// TIA Portal V17 export
// export: Created 2026-04-13T11:12:43.5748285Z, ExportSetting WithDefaults, DisplayName Totally Integrated Automation Portal, DisplayVersion V17 Update 4, DisplayName TIA Portal Openness, DisplayVersion V17 Update 4, DisplayName TIA Portal Version Control Interface, DisplayVersion V17, DisplayName SINAMICS Startdrive Advanced, DisplayVersion V17, DisplayName SINAMICS Startdrive G130, G150, S120, S150, SINAMICS MV, S210, DisplayVersion V17, DisplayName SINAMICS Startdrive G110M, G120, G120C, G120D, G120P, G115D, DisplayVersion V17, DisplayName STEP 7 Professional, DisplayVersion V17 Update 4, DisplayName STEP 7 Safety, DisplayVersion V17, DisplayName WinCC Professional, DisplayVersion V17 Update 4
FUNCTION_BLOCK "31-温度控制"   // FB21, LAD
{ S7_Optimized_Access := 'FALSE' }
VERSION : 0.1
// stored: AutoNumber true, IsIECCheckEnabled false, SetENOAutomatically false, UDAEnableTagReadback false
   VAR_IN_OUT
      进温设定 : Real;
      加热器开关 : Bool;
      自整定开关 : Bool;
      进温读 : Real;
      出温读 : Real;
      尾温读 : Real;
      进风温度P : Real;
      进风温度I : Real;
      进风温度D : Real;
      JF进风温度写读 : Real;
   END_VAR
   VAR DB_SPECIFIC
      CTU { S7_SetPoint := 'True'} : CTU_INT;
      TEMP { S7_SetPoint := 'True'} : Bool;
      TP : Array[0..40] of Bool;
      T1_PV_读 : Int;
      T2_PV_读 : Int;
      T3_PV_读 : Int;
      T4_PV_读 : Int;
      T5_PV_读 : Int;
      T1_SV_写 : Int;
      T1_P值比对1 : Int;
      T1_P值比对2 : Int;
      ST1 : Real;
      ST2 : Real;
      ST3 : Real;
      ST4 : Real;
      ST5 : Real;
      ST16 : Real;
      ST17 : Real;
      ST18 : Real;
      ST20 : Real;
      ST21 : Real;
      ST22 : Real;
      进温P读 : Int;
      进温I读 : Int;
      进温D读 : Int;
      T1_P_I_D_读 : Array[0..2] of Int;
      IEC_Timer_0_Instance { S7_SetPoint := 'True'} : TON_TIME;
      JF进风温度写读辅 { S7_SetPoint := 'True'} : Int;
      进温AT_写 : Int;
      进温AT_读 : Int;
      自整定开关字 : Int;
      加热器开关字 : Int;
   END_VAR
   VAR
      Modbus_Comm_Load_Instance { S7_SetPoint := 'True'} : Modbus_Comm_Load;
      Modbus_Master { S7_SetPoint := 'True'} : Modbus_Master;
   END_VAR
   VAR_TEMP   // added for the SCL form of the ladder/FBD networks
      _w1 : Bool;
      _w2 : Bool;
      _w3 : Bool;
      _w4 : Bool;
   END_VAR
BEGIN

REGION Network 1
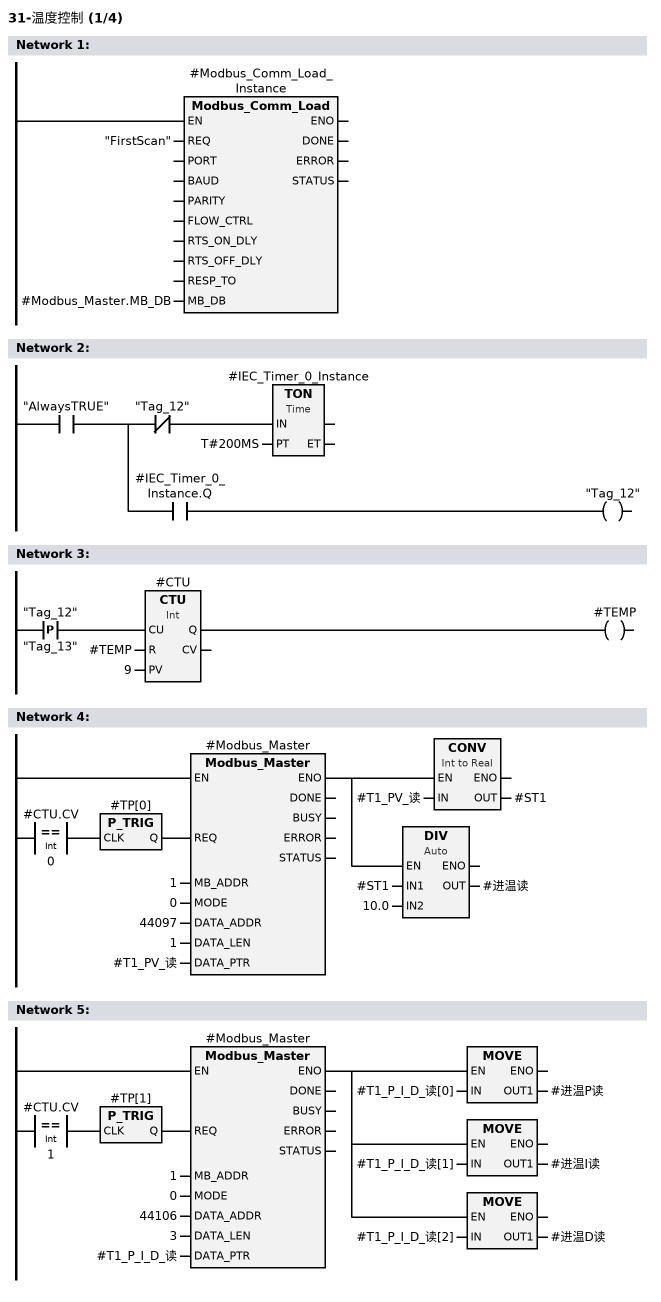
   RUNG wire#powerrail
      #Modbus_Comm_Load_Instance.Modbus_Comm_Load(REQ := "FirstScan", PORT :=, BAUD :=, PARITY :=, FLOW_CTRL :=, RTS_ON_DLY :=, RTS_OFF_DLY :=, RESP_TO :=, MB_DB := #Modbus_Master.MB_DB, DONE =>, ERROR =>, STATUS =>)
   END_RUNG
   // the same network as SCL:
   #Modbus_Comm_Load_Instance(REQ := "FirstScan", MB_DB := #Modbus_Master.MB_DB);   // Modbus_Comm_Load
END_REGION

REGION Network 2
   RUNG wire#powerrail
      Contact( "AlwaysTRUE" )
      wire#w1
      I_Contact( "Tag_12" )
      { S7_Templates := "time_type := Time" } #IEC_Timer_0_Instance.TON(pt := T#200MS, et =>)
   END_RUNG
   RUNG wire#w1
      Contact( #IEC_Timer_0_Instance.Q )
      Coil( "Tag_12" )
   END_RUNG
   // the same network as SCL:
   #IEC_Timer_0_Instance(IN := "AlwaysTRUE" AND NOT "Tag_12", PT := T#200MS);   // TON
   "Tag_12" := "AlwaysTRUE" AND #IEC_Timer_0_Instance.Q;
END_REGION

REGION Network 3
   RUNG wire#powerrail
      P_Contact(operand := "Tag_12", bit := "Tag_13")
      { S7_Templates := "value_type := Int" } #CTU.CTU(r := #TEMP, pv := 9, cv =>)
      Coil( #TEMP )
   END_RUNG
   // the same network as SCL:
   #_w1 := "Tag_12" AND NOT "Tag_13";   // rising edge of "Tag_12"
   "Tag_13" := "Tag_12";
   #CTU(CU := #_w1, R := #TEMP, PV := 9);   // CTU
   #TEMP := #CTU.Q;
END_REGION

REGION Network 4
   RUNG wire#powerrail
      #Modbus_Master.Modbus_Master(REQ := wire#w1, MB_ADDR := 1, MODE := 0, DATA_ADDR := 44097, DATA_LEN := 1, DATA_PTR := #T1_PV_读, DONE =>, BUSY =>, ERROR =>, STATUS =>)
      wire#w2
      { S7_Templates := "[SrcType := Int, DestType := Real]" } Convert(in := #T1_PV_读, out => #ST1)
   END_RUNG
   RUNG wire#powerrail
      { S7_Templates := "SrcType := Int" } EQ_Contact(in1 := #CTU.CV, in2 := 0)
      P_Trig( #TP[0] )
   END_RUNG wire#w1
   RUNG wire#w2
      Div(in1 := #ST1, in2 := 10.0, out => #进温读)
   END_RUNG
   // the same network as SCL:
   #_w1 := #CTU.CV = 0;
   #_w2 := #_w1 AND NOT #TP[0];   // rising edge
   #TP[0] := #_w1;
   #Modbus_Master(REQ := #_w2,   // Modbus_Master
                  MB_ADDR := 1,
                  MODE := 0,
                  DATA_ADDR := 44097,
                  DATA_LEN := 1,
                  DATA_PTR := #T1_PV_读,
                  ENO => #_w3);
   IF #_w3 THEN
       #ST1 := INT_TO_REAL(#T1_PV_读);
       #进温读 := #ST1 / 10.0;
   END_IF;
END_REGION

REGION Network 5
   RUNG wire#powerrail
      #Modbus_Master.Modbus_Master(REQ := wire#w1, MB_ADDR := 1, MODE := 0, DATA_ADDR := 44106, DATA_LEN := 3, DATA_PTR := #T1_P_I_D_读, DONE =>, BUSY =>, ERROR =>, STATUS =>)
      wire#w2
      Move(in := #T1_P_I_D_读[0], out1 => #进温P读)
   END_RUNG
   RUNG wire#powerrail
      { S7_Templates := "SrcType := Int" } EQ_Contact(in1 := #CTU.CV, in2 := 1)
      P_Trig( #TP[1] )
   END_RUNG wire#w1
   RUNG wire#w2
      Move(in := #T1_P_I_D_读[1], out1 => #进温I读)
   END_RUNG
   RUNG wire#w2
      Move(in := #T1_P_I_D_读[2], out1 => #进温D读)
   END_RUNG
   // the same network as SCL:
   #_w1 := #CTU.CV = 1;
   #_w2 := #_w1 AND NOT #TP[1];   // rising edge
   #TP[1] := #_w1;
   #Modbus_Master(REQ := #_w2,   // Modbus_Master
                  MB_ADDR := 1,
                  MODE := 0,
                  DATA_ADDR := 44106,
                  DATA_LEN := 3,
                  DATA_PTR := #T1_P_I_D_读,
                  ENO => #_w3);
   IF #_w3 THEN
       #进温P读 := #T1_P_I_D_读[0];
       #进温I读 := #T1_P_I_D_读[1];
       #进温D读 := #T1_P_I_D_读[2];
   END_IF;
END_REGION

REGION Network 6
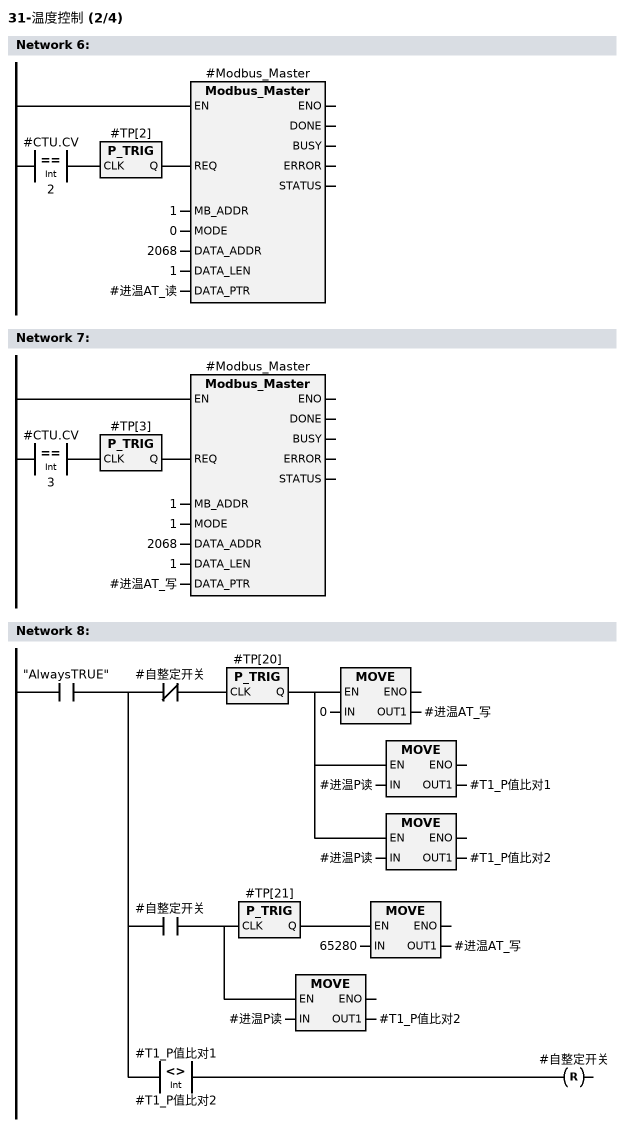
   RUNG wire#powerrail
      #Modbus_Master.Modbus_Master(REQ := wire#w1, MB_ADDR := 1, MODE := 0, DATA_ADDR := 2068, DATA_LEN := 1, DATA_PTR := #进温AT_读, DONE =>, BUSY =>, ERROR =>, STATUS =>)
   END_RUNG
   RUNG wire#powerrail
      { S7_Templates := "SrcType := Int" } EQ_Contact(in1 := #CTU.CV, in2 := 2)
      P_Trig( #TP[2] )
   END_RUNG wire#w1
   // the same network as SCL:
   #_w1 := #CTU.CV = 2;
   #_w2 := #_w1 AND NOT #TP[2];   // rising edge
   #TP[2] := #_w1;
   #Modbus_Master(REQ := #_w2, MB_ADDR := 1, MODE := 0, DATA_ADDR := 2068, DATA_LEN := 1, DATA_PTR := #进温AT_读);   // Modbus_Master
END_REGION

REGION Network 7
   RUNG wire#powerrail
      #Modbus_Master.Modbus_Master(REQ := wire#w1, MB_ADDR := 1, MODE := 1, DATA_ADDR := 2068, DATA_LEN := 1, DATA_PTR := #进温AT_写, DONE =>, BUSY =>, ERROR =>, STATUS =>)
   END_RUNG
   RUNG wire#powerrail
      { S7_Templates := "SrcType := Int" } EQ_Contact(in1 := #CTU.CV, in2 := 3)
      P_Trig( #TP[3] )
   END_RUNG wire#w1
   // the same network as SCL:
   #_w1 := #CTU.CV = 3;
   #_w2 := #_w1 AND NOT #TP[3];   // rising edge
   #TP[3] := #_w1;
   #Modbus_Master(REQ := #_w2, MB_ADDR := 1, MODE := 1, DATA_ADDR := 2068, DATA_LEN := 1, DATA_PTR := #进温AT_写);   // Modbus_Master
END_REGION

REGION Network 8
   RUNG wire#powerrail
      Contact( "AlwaysTRUE" )
      wire#w1
      I_Contact( #自整定开关 )
      P_Trig( #TP[20] )
      wire#w2
      Move(in := 0, out1 => #进温AT_写)
   END_RUNG
   RUNG wire#w2
      Move(in := #进温P读, out1 => #T1_P值比对1)
   END_RUNG
   RUNG wire#w2
      Move(in := #进温P读, out1 => #T1_P值比对2)
   END_RUNG
   RUNG wire#w1
      Contact( #自整定开关 )
      wire#w3
      P_Trig( #TP[21] )
      Move(in := 65280, out1 => #进温AT_写)
   END_RUNG
   RUNG wire#w3
      Move(in := #进温P读, out1 => #T1_P值比对2)
   END_RUNG
   RUNG wire#w1
      { S7_Templates := "SrcType := Int" } NE_Contact(in1 := #T1_P值比对1, in2 := #T1_P值比对2)
      R_Coil( #自整定开关 )
   END_RUNG
   // the same network as SCL:
   #_w1 := "AlwaysTRUE" AND NOT #自整定开关;
   #_w2 := #_w1 AND NOT #TP[20];   // rising edge
   #TP[20] := #_w1;
   IF #_w2 THEN
       #进温AT_写 := 0;
       #T1_P值比对1 := #进温P读;
       #T1_P值比对2 := #进温P读;
   END_IF;
   #_w3 := "AlwaysTRUE" AND #自整定开关;
   #_w4 := #_w3 AND NOT #TP[21];   // rising edge
   #TP[21] := #_w3;
   IF #_w4 THEN #进温AT_写 := 65280; END_IF;
   IF #_w3 THEN #T1_P值比对2 := #进温P读; END_IF;
   IF "AlwaysTRUE" AND (#T1_P值比对1 <> #T1_P值比对2) THEN #自整定开关 := FALSE; END_IF;
END_REGION

REGION Network 9
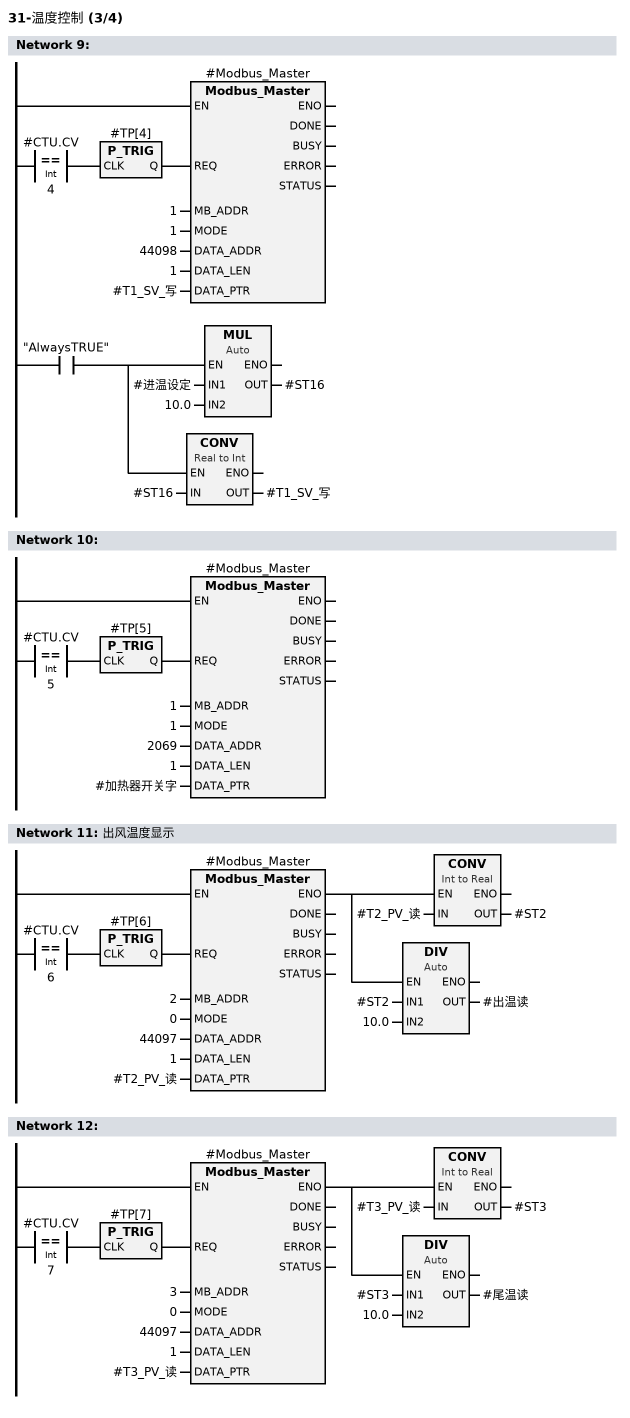
   RUNG wire#powerrail
      #Modbus_Master.Modbus_Master(REQ := wire#w1, MB_ADDR := 1, MODE := 1, DATA_ADDR := 44098, DATA_LEN := 1, DATA_PTR := #T1_SV_写, DONE =>, BUSY =>, ERROR =>, STATUS =>)
   END_RUNG
   RUNG wire#powerrail
      { S7_Templates := "SrcType := Int" } EQ_Contact(in1 := #CTU.CV, in2 := 4)
      P_Trig( #TP[4] )
   END_RUNG wire#w1
   RUNG wire#powerrail
      Contact( "AlwaysTRUE" )
      wire#w2
      Mul(in1 := #进温设定, in2 := 10.0, out => #ST16)
   END_RUNG
   RUNG wire#w2
      { S7_Templates := "[SrcType := Real, DestType := Int]" } Convert(in := #ST16, out => #T1_SV_写)
   END_RUNG
   // the same network as SCL:
   #_w1 := #CTU.CV = 4;
   #_w2 := #_w1 AND NOT #TP[4];   // rising edge
   #TP[4] := #_w1;
   #Modbus_Master(REQ := #_w2, MB_ADDR := 1, MODE := 1, DATA_ADDR := 44098, DATA_LEN := 1, DATA_PTR := #T1_SV_写);   // Modbus_Master
   IF "AlwaysTRUE" THEN
       #ST16 := #进温设定 * 10.0;
       #T1_SV_写 := REAL_TO_INT(#ST16);
   END_IF;
END_REGION

REGION Network 10
   RUNG wire#powerrail
      #Modbus_Master.Modbus_Master(REQ := wire#w1, MB_ADDR := 1, MODE := 1, DATA_ADDR := 2069, DATA_LEN := 1, DATA_PTR := #加热器开关字, DONE =>, BUSY =>, ERROR =>, STATUS =>)
   END_RUNG
   RUNG wire#powerrail
      { S7_Templates := "SrcType := Int" } EQ_Contact(in1 := #CTU.CV, in2 := 5)
      P_Trig( #TP[5] )
   END_RUNG wire#w1
   // the same network as SCL:
   #_w1 := #CTU.CV = 5;
   #_w2 := #_w1 AND NOT #TP[5];   // rising edge
   #TP[5] := #_w1;
   #Modbus_Master(REQ := #_w2, MB_ADDR := 1, MODE := 1, DATA_ADDR := 2069, DATA_LEN := 1, DATA_PTR := #加热器开关字);   // Modbus_Master
END_REGION

REGION Network 11: 出风温度显示
   RUNG wire#powerrail
      #Modbus_Master.Modbus_Master(REQ := wire#w1, MB_ADDR := 2, MODE := 0, DATA_ADDR := 44097, DATA_LEN := 1, DATA_PTR := #T2_PV_读, DONE =>, BUSY =>, ERROR =>, STATUS =>)
      wire#w2
      { S7_Templates := "[SrcType := Int, DestType := Real]" } Convert(in := #T2_PV_读, out => #ST2)
   END_RUNG
   RUNG wire#powerrail
      { S7_Templates := "SrcType := Int" } EQ_Contact(in1 := #CTU.CV, in2 := 6)
      P_Trig( #TP[6] )
   END_RUNG wire#w1
   RUNG wire#w2
      Div(in1 := #ST2, in2 := 10.0, out => #出温读)
   END_RUNG
   // the same network as SCL:
   #_w1 := #CTU.CV = 6;
   #_w2 := #_w1 AND NOT #TP[6];   // rising edge
   #TP[6] := #_w1;
   #Modbus_Master(REQ := #_w2,   // Modbus_Master
                  MB_ADDR := 2,
                  MODE := 0,
                  DATA_ADDR := 44097,
                  DATA_LEN := 1,
                  DATA_PTR := #T2_PV_读,
                  ENO => #_w3);
   IF #_w3 THEN
       #ST2 := INT_TO_REAL(#T2_PV_读);
       #出温读 := #ST2 / 10.0;
   END_IF;
END_REGION

REGION Network 12
   RUNG wire#powerrail
      #Modbus_Master.Modbus_Master(REQ := wire#w1, MB_ADDR := 3, MODE := 0, DATA_ADDR := 44097, DATA_LEN := 1, DATA_PTR := #T3_PV_读, DONE =>, BUSY =>, ERROR =>, STATUS =>)
      wire#w2
      { S7_Templates := "[SrcType := Int, DestType := Real]" } Convert(in := #T3_PV_读, out => #ST3)
   END_RUNG
   RUNG wire#powerrail
      { S7_Templates := "SrcType := Int" } EQ_Contact(in1 := #CTU.CV, in2 := 7)
      P_Trig( #TP[7] )
   END_RUNG wire#w1
   RUNG wire#w2
      Div(in1 := #ST3, in2 := 10.0, out => #尾温读)
   END_RUNG
   // the same network as SCL:
   #_w1 := #CTU.CV = 7;
   #_w2 := #_w1 AND NOT #TP[7];   // rising edge
   #TP[7] := #_w1;
   #Modbus_Master(REQ := #_w2,   // Modbus_Master
                  MB_ADDR := 3,
                  MODE := 0,
                  DATA_ADDR := 44097,
                  DATA_LEN := 1,
                  DATA_PTR := #T3_PV_读,
                  ENO => #_w3);
   IF #_w3 THEN
       #ST3 := INT_TO_REAL(#T3_PV_读);
       #尾温读 := #ST3 / 10.0;
   END_IF;
END_REGION

REGION Network 13
   // 冷水机温du
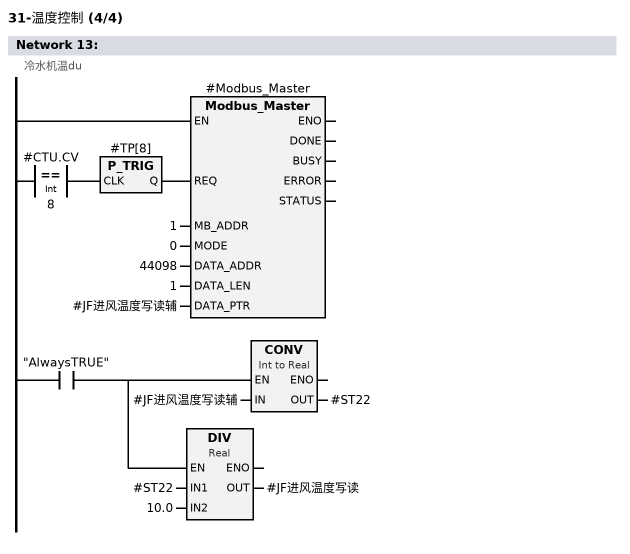
   RUNG wire#powerrail
      #Modbus_Master.Modbus_Master(REQ := wire#w1, MB_ADDR := 1, MODE := 0, DATA_ADDR := 44098, DATA_LEN := 1, DATA_PTR := #JF进风温度写读辅, DONE =>, BUSY =>, ERROR =>, STATUS =>)
   END_RUNG
   RUNG wire#powerrail
      { S7_Templates := "SrcType := Int" } EQ_Contact(in1 := #CTU.CV, in2 := 8)
      P_Trig( #TP[8] )
   END_RUNG wire#w1
   RUNG wire#powerrail
      Contact( "AlwaysTRUE" )
      wire#w2
      { S7_Templates := "[SrcType := Int, DestType := Real]" } Convert(in := #JF进风温度写读辅, out => #ST22)
   END_RUNG
   RUNG wire#w2
      { S7_Templates := "SrcType := Real" } Div(in1 := #ST22, in2 := 10.0, out => #JF进风温度写读)
   END_RUNG
   // the same network as SCL:
   #_w1 := #CTU.CV = 8;
   #_w2 := #_w1 AND NOT #TP[8];   // rising edge
   #TP[8] := #_w1;
   #Modbus_Master(REQ := #_w2,   // Modbus_Master
                  MB_ADDR := 1,
                  MODE := 0,
                  DATA_ADDR := 44098,
                  DATA_LEN := 1,
                  DATA_PTR := #JF进风温度写读辅);
   IF "AlwaysTRUE" THEN
       #ST22 := INT_TO_REAL(#JF进风温度写读辅);
       #JF进风温度写读 := #ST22 / 10.0;
   END_IF;
END_REGION

REGION Network 14 (SCL)
   #进风温度P := INT_TO_REAL(#进温P读);
   #进风温度I := INT_TO_REAL(#进温I读);
   #进风温度D := INT_TO_REAL(#进温D读);
   IF #加热器开关 THEN
       #加热器开关字 := 65280;
   ELSE
       #加热器开关字 := 0;
   END_IF;
END_REGION
END_FUNCTION_BLOCK
